{attribute addProperty BoxType "EP2809-0042-0018"}
{attribute addProperty Id "DO_X01AT %Q*ARRAY[0..1] OF DO_X_7F374EB0429496728842949672950DO_X02AT %Q*ARRAY[0..1] OF DO_X_7F374EB0429496728842949672950DO_X03AT %Q*ARRAY[0..1] OF DO_X_7F374EB0429496728842949672950DO_X04AT %Q*ARRAY[0..1] OF DO_X_7F374EB0429496728842949672950DO_X05AT %Q*ARRAY[0..1] OF DO_X_7F374EB0429496728842949672950DO_X06AT %Q*ARRAY[0..1] OF DO_X_7F374EB0429496728842949672950DO_X07AT %Q*ARRAY[0..1] OF DO_X_7F374EB0429496728842949672950DO_X08AT %Q*ARRAY[0..1] OF DO_X_7F374EB0429496728842949672950WcStateAT %I*WcState_28A8677510.1250InfoDataAT %I*InfoData_192954DE1620"}
{attribute addProperty CRC "3861973089"}
{attribute addProperty SizeInBites "4294967249"}
{attribute addProperty SizeInBytes "34359738362.125"}
TYPE EP2809_556C4F60 :
STRUCT
	{attribute addProperty Name "DO_X01"}
	DO_X01 : ARRAY[0..1] OF DO_X_7F374EB0;
	{attribute addProperty Name "DO_X02"}
	DO_X02 : ARRAY[0..1] OF DO_X_7F374EB0;
	{attribute addProperty Name "DO_X03"}
	DO_X03 : ARRAY[0..1] OF DO_X_7F374EB0;
	{attribute addProperty Name "DO_X04"}
	DO_X04 : ARRAY[0..1] OF DO_X_7F374EB0;
	{attribute addProperty Name "DO_X05"}
	DO_X05 : ARRAY[0..1] OF DO_X_7F374EB0;
	{attribute addProperty Name "DO_X06"}
	DO_X06 : ARRAY[0..1] OF DO_X_7F374EB0;
	{attribute addProperty Name "DO_X07"}
	DO_X07 : ARRAY[0..1] OF DO_X_7F374EB0;
	{attribute addProperty Name "DO_X08"}
	DO_X08 : ARRAY[0..1] OF DO_X_7F374EB0;
	{attribute addProperty Name "WcState"}
	WcState : WcState_28A86775;
	{attribute addProperty Name "InfoData"}
	InfoData : InfoData_192954DE;
END_STRUCT
END_TYPE

(* stored: Version 1.2.0.0, ProductVersion 3.1.4024.9
   DUT EP2809_556C4F60: Id {8e6e720d-89cf-4e77-b4ea-23ede0cc5bf7} *)
